FUNCTION_BLOCK FB_ReservoirHeaterIsOn
VAR_INPUT
	ReservoirTemperature : REAL ; // Celcius
	ReservoirHeaterIsOn : BOOL ; 
	ReservoirHeaterSPon : REAL ; // Celcius
	ReservoirHeaterSPoff : REAL ; // Celcius
	BoolSimulationTesting : BOOL ; //True if testing with PLC logic
END_VAR

IF NOT BoolSimulationTesting THEN
	IF (ReservoirTemperature < ReservoirHeaterSPon) THEN
		ReservoirHeaterIsOn := TRUE ; 
	ELSIF ((ReservoirTemperature > ReservoirHeaterSPon) AND (ReservoirTemperature < ReservoirHeaterSPoff)) AND ReservoirHeaterIsOn THEN
		ReservoirHeaterIsOn :=TRUE; 
	ELSIF ((ReservoirTemperature > ReservoirHeaterSPon) AND (ReservoirTemperature < ReservoirHeaterSPoff)) AND NOT ReservoirHeaterIsOn THEN
		ReservoirHeaterIsOn :=FALSE;
	ELSIF (ReservoirTemperature > ReservoirHeaterSPoff) THEN
		ReservoirHeaterIsOn :=FALSE;
	END_IF
END_IF

END_FUNCTION_BLOCK

(* stored: Version 1.1.0.1, ProductVersion 3.1.4024.12
   POU FB_ReservoirHeaterIsOn: Id {5134fce4-4bf6-4059-be17-cc9309695c95}, SpecialFunc None *)
